TYPE WheelVelocity :
STRUCT
	wheel1, wheel2, wheel3 : LREAL;
END_STRUCT
END_TYPE

(* stored: Version 1.1.0.1, ProductVersion 3.1.4026.13
   DUT WheelVelocity: Id {86fa5370-f65a-40c4-9bdd-46f82ebb81f1} *)
